FUNCTION_BLOCK CallButton_HMI (* Service Interface Function Block Type *)
  (* Standard: 61499-2 *)
  (* Version 0.0, 6/3/2016, Andrei, nxtControl GmbH, template *)
  PACKAGE Main;
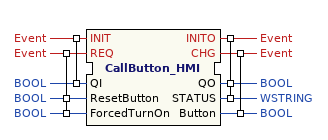
  EVENT_INPUT
    INIT WITH QI;
    REQ WITH ResetButton, ForcedTurnOn;
  END_EVENT
  EVENT_OUTPUT
    INITO WITH QO, STATUS;
    CHG WITH Button;
  END_EVENT
  VAR_INPUT
    QI : BOOL;
    ResetButton : BOOL;
    ForcedTurnOn : BOOL;
  END_VAR
  VAR_OUTPUT
    QO : BOOL; (* Event Output Qualifier *)
    STATUS : WSTRING; (* Service Status *)
    Button : BOOL;
  END_VAR
END_FUNCTION_BLOCK
